{attribute 'qualified_only'}
{attribute 'strict'}
{attribute 'to_string'}
TYPE E_St030_EmptySlotChk :
(
	eSt030_EmptySlotChk_none := 0,
	eSt030_EmptySlotChk_Empty,
	eSt030_EmptySlotChk_NotEmpty
);
END_TYPE

(* stored: Version 1.1.0.1
   DUT E_St030_EmptySlotChk: Id {c1c0c076-d4b6-40c1-a8f2-4242acf45b37} *)
